(* IEC 61131-3 sources: Std_PalletMover/Class/Curtis_AC2F_IO, 1 file *)

(* ---- Curtis_AC2F_IO.st ---- *)
(*!
<Class
	Name               = "Curtis_AC2F_IO"
	Revision           = "0.0"
	RealtimeTask       = "false"
	CyclicTask         = "false"
	BackgroundTask     = "false"
	Sigmatek           = "false"
	OSInterface        = "false"
	HighPriority       = "false"
	Automatic          = "false"
	UpdateMode         = "Prescan"
	SharedCommandTable = "true"
	Objectsize         = "(570,1380)">
	<Channels>
		<Server Name="ClassSvr" Visualized="false" Initialize="false" WriteProtected="true" Retentive="false"/>
		<Server Name="In11_Enc1_c" Visualized="false" Initialize="false" WriteProtected="true" Retentive="false"/>
		<Server Name="In12" Visualized="false" Initialize="false" WriteProtected="true" Retentive="false"/>
		<Server Name="In13" Visualized="false" Initialize="false" WriteProtected="true" Retentive="false"/>
		<Server Name="In14_An14" Visualized="false" Initialize="false" WriteProtected="true" Retentive="false"/>
		<Server Name="In1_An1" Visualized="false" Initialize="false" WriteProtected="true" Retentive="false"/>
		<Server Name="In2_An2_Temp" Visualized="false" Initialize="false" WriteProtected="true" Retentive="false"/>
		<Server Name="In5_An5" Visualized="false" Initialize="false" WriteProtected="true" Retentive="false"/>
		<Server Name="In6_An6" Visualized="false" Initialize="false" WriteProtected="true" Retentive="false" Comment="Pin10"/>
		<Server Name="In7_An7" Visualized="false" Initialize="false" WriteProtected="true" Retentive="false"/>
		<Server Name="In8_An8" Visualized="false" Initialize="false" WriteProtected="true" Retentive="false"/>
		<Server Name="Out1_In21" Visualized="true" Initialize="false" WriteProtected="false" Retentive="false"/>
		<Server Name="Out2_In22" Visualized="true" Initialize="false" WriteProtected="false" Retentive="false"/>
		<Server Name="Out3_In23" Visualized="true" Initialize="false" WriteProtected="false" Retentive="false"/>
		<Server Name="Out4_In24" Visualized="true" Initialize="false" WriteProtected="false" Retentive="false"/>
		<Server Name="Out5_In25" Visualized="true" Initialize="false" WriteProtected="false" Retentive="false"/>
		<Server Name="Out_ResetEm" Visualized="true" Initialize="false" WriteProtected="false" Retentive="false"/>
		<Server Name="xIn21" Visualized="false" Initialize="false" WriteProtected="true" Retentive="false"/>
		<Server Name="xIn22" Visualized="false" Initialize="false" WriteProtected="true" Retentive="false"/>
		<Server Name="xIn23" Visualized="false" Initialize="false" WriteProtected="true" Retentive="false"/>
		<Server Name="xIn24" Visualized="false" Initialize="false" WriteProtected="true" Retentive="false"/>
		<Server Name="xIn25" Visualized="false" Initialize="false" WriteProtected="true" Retentive="false"/>
	</Channels>
</Class>
*)
Curtis_AC2F_IO : CLASS
  //Servers:
	ClassSvr 	: SvrChCmd_DINT;
	In14_An14 	: SvrCh_DINT;
	In13 	: SvrCh_DINT;
	In12 	: SvrCh_DINT;
	In11_Enc1_c 	: SvrCh_DINT;
	In8_An8 	: SvrCh_DINT;
	In7_An7 	: SvrCh_DINT;
	In5_An5 	: SvrCh_DINT;
	In6_An6 	: SvrCh_DINT;
	In1_An1 	: SvrCh_DINT;
	In2_An2_Temp 	: SvrCh_DINT;
	Out3_In23 	: SvrCh_DINT;
	xIn23 	: SvrCh_DINT;
	Out2_In22 	: SvrCh_DINT;
	xIn22 	: SvrCh_DINT;
	Out5_In25 	: SvrCh_DINT;
	xIn25 	: SvrCh_DINT;
	Out4_In24 	: SvrCh_DINT;
	xIn24 	: SvrCh_DINT;
	Out1_In21 	: SvrCh_DINT;
	xIn21 	: SvrCh_DINT;
	Out_ResetEm 	: SvrCh_DINT;
  //Clients:
  //Variables:
  //Functions:

	FUNCTION GLOBAL UpdateInput
		VAR_INPUT
			pdoSplitOut1 	: BSINT;
			pdoSplitOut2 	: BSINT;
		END_VAR;

	FUNCTION GLOBAL UpdateOutput
		VAR_OUTPUT
			outBDINT 	: BINT;
		END_VAR;
  //Tables:
	FUNCTION @STD
		VAR_OUTPUT
			ret_code	: CONFSTATES;
		END_VAR;
	FUNCTION GLOBAL TAB @CT_;
END_CLASS;

FUNCTION GLOBAL Curtis_AC2F_IO::UpdateInput
	VAR_INPUT
		pdoSplitOut1 	: BSINT;
		pdoSplitOut2 	: BSINT;
	END_VAR

    //----------------------------------------------------
  // Read out PDO_RX3 with identifier 0x380 + NodeID
  //----------------------------------------------------

    In1_An1         := pdoSplitOut1.1;
    In2_An2_Temp    := pdoSplitOut1.2;
    //pdoSplitOut1.3
    //pdoSplitOut1.4
    In5_An5         := pdoSplitOut1.5;
    In6_An6         := pdoSplitOut1.6;
    In7_An7         := pdoSplitOut1.7;
    In8_An8         := pdoSplitOut1.8;
    //pdoSplitOut2.1;
    //pdoSplitOut2.2;

    In11_Enc1_c     := pdoSplitOut2.3;
    In12            := pdoSplitOut2.4;
    In13            := pdoSplitOut2.5;
    In14_An14       := pdoSplitOut2.6;

   (*xIn23           := pdoSplitOut2.4;
    xIn22           := pdoSplitOut2.3;
    xIn25           := pdoSplitOut2.5;
    xIn24           := pdoSplitOut2.6;
    xIn21           := pdoSplitOut2.7;
    *)

END_FUNCTION

FUNCTION GLOBAL Curtis_AC2F_IO::UpdateOutput
	VAR_OUTPUT
		outBDINT 	: BINT;
	END_VAR

    outBDINT.1 := Out1_In21$bool;
    outBDINT.2 := Out2_In22$bool;
    outBDINT.3 := Out3_In23$bool;
    outBDINT.4 := Out4_In24$bool;
    outBDINT.5 := Out5_In25$bool;
    outBDINT.6 := Out_ResetEm$bool;
    outBDINT.7 := False;
    outBDINT.8 := False;
    outBDINT.9 := False;
    outBDINT.10 := False;
    outBDINT.11 := False;
    outBDINT.12 := False;
    outBDINT.13 := False;
    outBDINT.14 := False;
    outBDINT.15 := False;
    outBDINT.16 := False;

END_FUNCTION
